// TIA Portal project "Styringsenhed" (V13)

(* hardware
DEVICE "S7-1200 station_1"  S7-1200 Station
   slot 0: "Rack_0"  Rack  V1.0
   slot 1: "PLC_1"  CPU 1214C DC/DC/DC  6ES7 214-1AG40-0XB0  V4.1
   slot 3: "AQ 1x12BIT_1"  6ES7 232-4HA30-0XB0  V1.0
DEVICE "HMI_1"  KTP600 Basic color PN
   slot 0: "HMI"  HMI  6AV6 647-0AD11-3AX0  12.0.0.0
   slot 1: "HMI_RT_1"  KTP600 Basic color PN  6AV6 647-0AD11-3AX0  12.0.0.0
   slot 5: "HMI_1.IE_CP_1"  PROFINET Interface
      slot 1: "PROFINET Interface_1"  PROFINET Interface
         slot 1: "Port_1"  Port
*)

// ===== PLC "PLC_1"  CPU 1214C DC/DC/DC =====

VAR_GLOBAL   // PLC tag table "Default tag table"
   "Trin1" AT %Q0.6 : Bool;
   "Trin2" AT %Q0.7 : Bool;
   "Trin3" AT %Q1.0 : Bool;
   "Trin4" AT %Q1.1 : Bool;
   "SpændingCentral" AT %MB0 : USInt;
   "ManuelMode" AT %I0.0 : Bool;
   "KnapOp" AT %I0.1 : Bool;
   "KnapNed" AT %I0.2 : Bool;
END_VAR

DATA_BLOCK "Trinskifter_DB"   // DB8
{ S7_Optimized_Access := 'FALSE' }
VERSION : 0.1
// stored: InstanceOfName Trinskifter
"Trinskifter"
BEGIN
END_DATA_BLOCK

// folder: System blocks/Program resources

DATA_BLOCK "ManTrinskift1til2"   // DB1
{ S7_Optimized_Access := 'FALSE' }
AUTHOR : Simatic
FAMILY : IEC
NAME : IEC_TMR
VERSION : 1.0
// stored: InstanceOfName ?
"?"
BEGIN
END_DATA_BLOCK

DATA_BLOCK "Trinskift2til1"   // DB2
{ S7_Optimized_Access := 'FALSE' }
AUTHOR : Simatic
FAMILY : IEC
NAME : IEC_TMR
VERSION : 1.0
// stored: InstanceOfName ?
"?"
BEGIN
END_DATA_BLOCK

DATA_BLOCK "Trinskift2til3"   // DB3
{ S7_Optimized_Access := 'FALSE' }
AUTHOR : Simatic
FAMILY : IEC
NAME : IEC_TMR
VERSION : 1.0
// stored: InstanceOfName ?
"?"
BEGIN
END_DATA_BLOCK

DATA_BLOCK "Trinskift1til2"   // DB4
{ S7_Optimized_Access := 'FALSE' }
AUTHOR : Simatic
FAMILY : IEC
NAME : IEC_TMR
VERSION : 1.0
// stored: InstanceOfName ?
"?"
BEGIN
END_DATA_BLOCK

DATA_BLOCK "Trinskift3til2"   // DB5
{ S7_Optimized_Access := 'FALSE' }
AUTHOR : Simatic
FAMILY : IEC
NAME : IEC_TMR
VERSION : 1.0
// stored: InstanceOfName ?
"?"
BEGIN
END_DATA_BLOCK

DATA_BLOCK "Trinskift3til4"   // DB6
{ S7_Optimized_Access := 'FALSE' }
AUTHOR : Simatic
FAMILY : IEC
NAME : IEC_TMR
VERSION : 1.0
// stored: InstanceOfName ?
"?"
BEGIN
END_DATA_BLOCK

DATA_BLOCK "Trinskift4til3"   // DB7
{ S7_Optimized_Access := 'FALSE' }
AUTHOR : Simatic
FAMILY : IEC
NAME : IEC_TMR
VERSION : 1.0
// stored: InstanceOfName ?
"?"
BEGIN
END_DATA_BLOCK

DATA_BLOCK "ManTrinskift2til3"   // DB9
{ S7_Optimized_Access := 'FALSE' }
AUTHOR : Simatic
FAMILY : IEC
NAME : IEC_TMR
VERSION : 1.0
// stored: InstanceOfName ?
"?"
BEGIN
END_DATA_BLOCK

DATA_BLOCK "ManTrinskift2til1"   // DB10
{ S7_Optimized_Access := 'FALSE' }
AUTHOR : Simatic
FAMILY : IEC
NAME : IEC_TMR
VERSION : 1.0
// stored: InstanceOfName ?
"?"
BEGIN
END_DATA_BLOCK

DATA_BLOCK "ManTrinskift3til4"   // DB11
{ S7_Optimized_Access := 'FALSE' }
AUTHOR : Simatic
FAMILY : IEC
NAME : IEC_TMR
VERSION : 1.0
// stored: InstanceOfName ?
"?"
BEGIN
END_DATA_BLOCK

DATA_BLOCK "ManTrinskift3til2"   // DB12
{ S7_Optimized_Access := 'FALSE' }
AUTHOR : Simatic
FAMILY : IEC
NAME : IEC_TMR
VERSION : 1.0
// stored: InstanceOfName ?
"?"
BEGIN
END_DATA_BLOCK

DATA_BLOCK "ManTrinskift4til3"   // DB13
{ S7_Optimized_Access := 'FALSE' }
AUTHOR : Simatic
FAMILY : IEC
NAME : IEC_TMR
VERSION : 1.0
// stored: InstanceOfName ?
"?"
BEGIN
END_DATA_BLOCK

// folder: (top level)

FUNCTION_BLOCK "Trinskifter"   // FB1, LAD
{ S7_Optimized_Access := 'FALSE' }
VERSION : 0.1
   VAR_TEMP   // added for the SCL form of the ladder/FBD networks
      _w1 : Bool;
      _w2 : Bool;
   END_VAR
BEGIN

REGION Network 1: Start
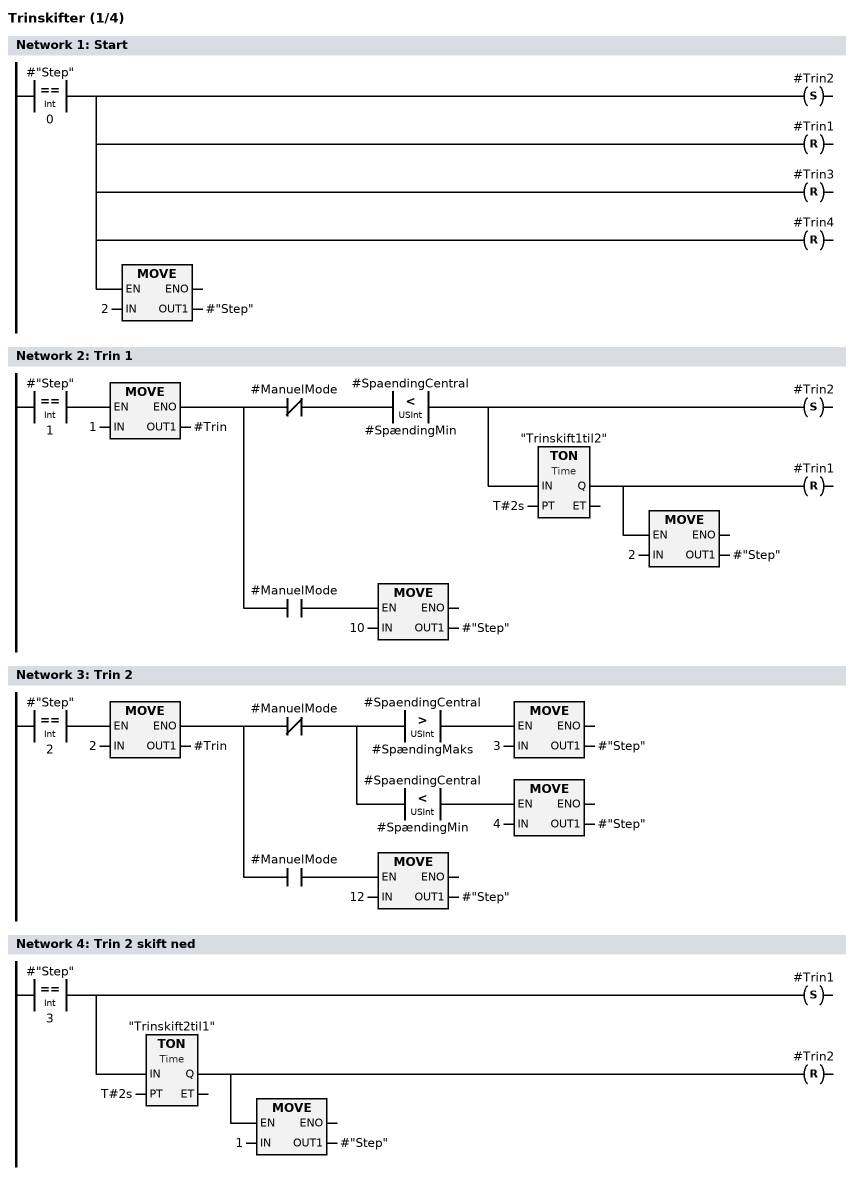
   RUNG wire#powerrail
      { S7_Templates := "SrcType := Int" } EQ_Contact(in1 := #"Step", in2 := 0)
      wire#w1
      S_Coil( #Trin2 )
   END_RUNG
   RUNG wire#w1
      R_Coil( #Trin1 )
   END_RUNG
   RUNG wire#w1
      R_Coil( #Trin3 )
   END_RUNG
   RUNG wire#w1
      R_Coil( #Trin4 )
   END_RUNG
   RUNG wire#w1
      Move(in := 2, out1 => #"Step")
   END_RUNG
   // the same network as SCL:
   IF #"Step" = 0 THEN
       #Trin2 := TRUE;
       #Trin1 := FALSE;
       #Trin3 := FALSE;
       #Trin4 := FALSE;
       #"Step" := 2;
   END_IF;
END_REGION

REGION Network 2: Trin 1
   #_w1 := #"Step" = 1;
   IF #_w1 THEN #Trin := 1; END_IF;
   #_w2 := #_w1 AND NOT #ManuelMode AND (#SpaendingCentral < #SpændingMin);
   IF #_w2 THEN #Trin2 := TRUE; END_IF;
   "Trinskift1til2".TON(IN := #_w2, PT := T#2s);
   IF "Trinskift1til2".Q THEN
       #Trin1 := FALSE;
       #"Step" := 2;
   END_IF;
   IF #_w1 AND #ManuelMode THEN #"Step" := 10; END_IF;
END_REGION

REGION Network 3: Trin 2
   RUNG wire#powerrail
      { S7_Templates := "SrcType := Int" } EQ_Contact(in1 := #"Step", in2 := 2)
      Move(in := 2, out1 => #Trin)
      wire#w1
      I_Contact( #ManuelMode )
      wire#w2
      { S7_Templates := "SrcType := USInt" } GT_Contact(in1 := #SpaendingCentral, in2 := #SpændingMaks)
      Move(in := 3, out1 => #"Step")
   END_RUNG
   RUNG wire#w2
      { S7_Templates := "SrcType := USInt" } LT_Contact(in1 := #SpaendingCentral, in2 := #SpændingMin)
      Move(in := 4, out1 => #"Step")
   END_RUNG
   RUNG wire#w1
      Contact( #ManuelMode )
      Move(in := 12, out1 => #"Step")
   END_RUNG
   // the same network as SCL:
   #_w1 := #"Step" = 2;
   IF #_w1 THEN #Trin := 2; END_IF;
   #_w2 := #_w1 AND NOT #ManuelMode;
   IF #_w2 AND (#SpaendingCentral > #SpændingMaks) THEN #"Step" := 3; END_IF;
   IF #_w2 AND (#SpaendingCentral < #SpændingMin) THEN #"Step" := 4; END_IF;
   IF #_w1 AND #ManuelMode THEN #"Step" := 12; END_IF;
END_REGION

REGION Network 4: Trin 2 skift ned
   #_w1 := #"Step" = 3;
   IF #_w1 THEN #Trin1 := TRUE; END_IF;
   "Trinskift2til1".TON(IN := #_w1, PT := T#2s);
   IF "Trinskift2til1".Q THEN
       #Trin2 := FALSE;
       #"Step" := 1;
   END_IF;
END_REGION

REGION Network 5: Trin 2 skift op
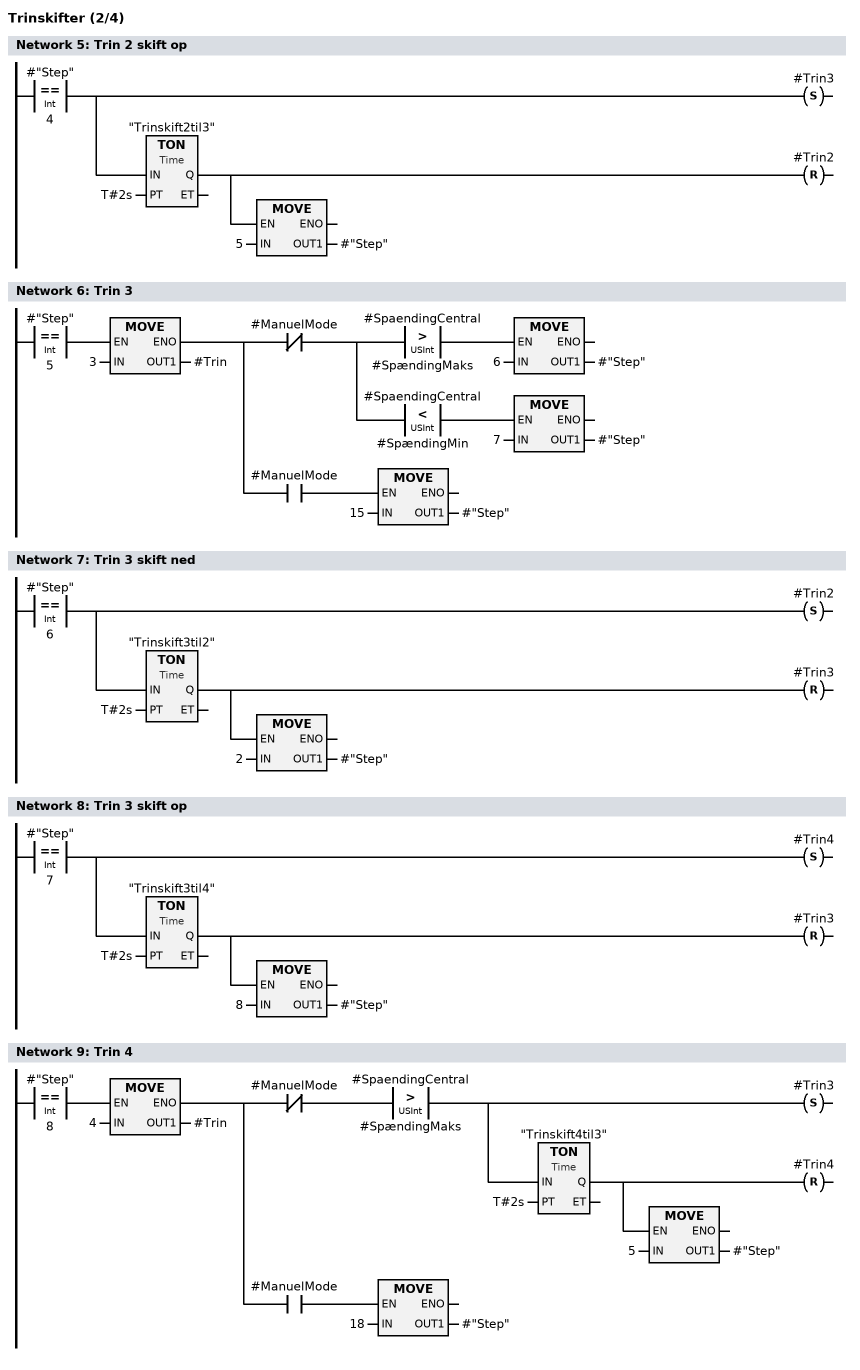
   #_w1 := #"Step" = 4;
   IF #_w1 THEN #Trin3 := TRUE; END_IF;
   "Trinskift2til3".TON(IN := #_w1, PT := T#2s);
   IF "Trinskift2til3".Q THEN
       #Trin2 := FALSE;
       #"Step" := 5;
   END_IF;
END_REGION

REGION Network 6: Trin 3
   RUNG wire#powerrail
      { S7_Templates := "SrcType := Int" } EQ_Contact(in1 := #"Step", in2 := 5)
      Move(in := 3, out1 => #Trin)
      wire#w1
      I_Contact( #ManuelMode )
      wire#w2
      { S7_Templates := "SrcType := USInt" } GT_Contact(in1 := #SpaendingCentral, in2 := #SpændingMaks)
      Move(in := 6, out1 => #"Step")
   END_RUNG
   RUNG wire#w2
      { S7_Templates := "SrcType := USInt" } LT_Contact(in1 := #SpaendingCentral, in2 := #SpændingMin)
      Move(in := 7, out1 => #"Step")
   END_RUNG
   RUNG wire#w1
      Contact( #ManuelMode )
      Move(in := 15, out1 => #"Step")
   END_RUNG
   // the same network as SCL:
   #_w1 := #"Step" = 5;
   IF #_w1 THEN #Trin := 3; END_IF;
   #_w2 := #_w1 AND NOT #ManuelMode;
   IF #_w2 AND (#SpaendingCentral > #SpændingMaks) THEN #"Step" := 6; END_IF;
   IF #_w2 AND (#SpaendingCentral < #SpændingMin) THEN #"Step" := 7; END_IF;
   IF #_w1 AND #ManuelMode THEN #"Step" := 15; END_IF;
END_REGION

REGION Network 7: Trin 3 skift ned
   #_w1 := #"Step" = 6;
   IF #_w1 THEN #Trin2 := TRUE; END_IF;
   "Trinskift3til2".TON(IN := #_w1, PT := T#2s);
   IF "Trinskift3til2".Q THEN
       #Trin3 := FALSE;
       #"Step" := 2;
   END_IF;
END_REGION

REGION Network 8: Trin 3 skift op
   #_w1 := #"Step" = 7;
   IF #_w1 THEN #Trin4 := TRUE; END_IF;
   "Trinskift3til4".TON(IN := #_w1, PT := T#2s);
   IF "Trinskift3til4".Q THEN
       #Trin3 := FALSE;
       #"Step" := 8;
   END_IF;
END_REGION

REGION Network 9: Trin 4
   #_w1 := #"Step" = 8;
   IF #_w1 THEN #Trin := 4; END_IF;
   #_w2 := #_w1 AND NOT #ManuelMode AND (#SpaendingCentral > #SpændingMaks);
   IF #_w2 THEN #Trin3 := TRUE; END_IF;
   "Trinskift4til3".TON(IN := #_w2, PT := T#2s);
   IF "Trinskift4til3".Q THEN
       #Trin4 := FALSE;
       #"Step" := 5;
   END_IF;
   IF #_w1 AND #ManuelMode THEN #"Step" := 18; END_IF;
END_REGION

REGION Network 10: Manuel trin 1
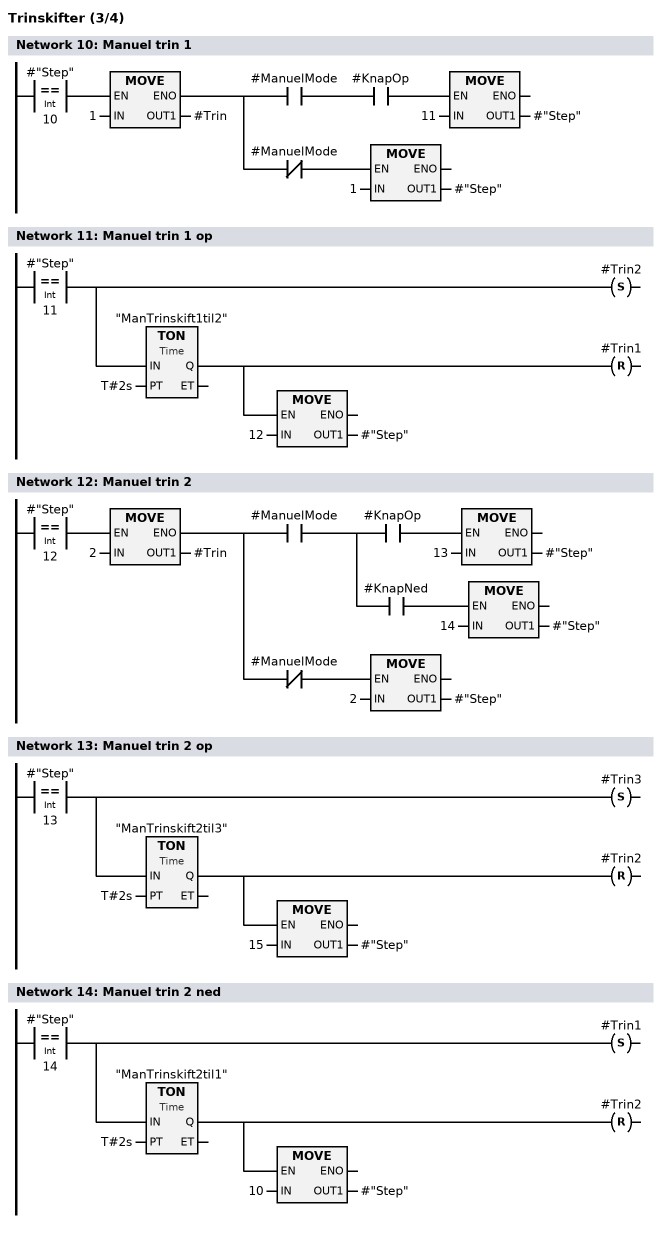
   RUNG wire#powerrail
      { S7_Templates := "SrcType := Int" } EQ_Contact(in1 := #"Step", in2 := 10)
      Move(in := 1, out1 => #Trin)
      wire#w1
      Contact( #ManuelMode )
      Contact( #KnapOp )
      Move(in := 11, out1 => #"Step")
   END_RUNG
   RUNG wire#w1
      I_Contact( #ManuelMode )
      Move(in := 1, out1 => #"Step")
   END_RUNG
   // the same network as SCL:
   #_w1 := #"Step" = 10;
   IF #_w1 THEN #Trin := 1; END_IF;
   IF #_w1 AND #ManuelMode AND #KnapOp THEN #"Step" := 11; END_IF;
   IF #_w1 AND NOT #ManuelMode THEN #"Step" := 1; END_IF;
END_REGION

REGION Network 11: Manuel trin 1 op
   #_w1 := #"Step" = 11;
   IF #_w1 THEN #Trin2 := TRUE; END_IF;
   "ManTrinskift1til2".TON(IN := #_w1, PT := T#2s);
   IF "ManTrinskift1til2".Q THEN
       #Trin1 := FALSE;
       #"Step" := 12;
   END_IF;
END_REGION

REGION Network 12: Manuel trin 2
   RUNG wire#powerrail
      { S7_Templates := "SrcType := Int" } EQ_Contact(in1 := #"Step", in2 := 12)
      Move(in := 2, out1 => #Trin)
      wire#w1
      Contact( #ManuelMode )
      wire#w2
      Contact( #KnapOp )
      Move(in := 13, out1 => #"Step")
   END_RUNG
   RUNG wire#w2
      Contact( #KnapNed )
      Move(in := 14, out1 => #"Step")
   END_RUNG
   RUNG wire#w1
      I_Contact( #ManuelMode )
      Move(in := 2, out1 => #"Step")
   END_RUNG
   // the same network as SCL:
   #_w1 := #"Step" = 12;
   IF #_w1 THEN #Trin := 2; END_IF;
   #_w2 := #_w1 AND #ManuelMode;
   IF #_w2 AND #KnapOp THEN #"Step" := 13; END_IF;
   IF #_w2 AND #KnapNed THEN #"Step" := 14; END_IF;
   IF #_w1 AND NOT #ManuelMode THEN #"Step" := 2; END_IF;
END_REGION

REGION Network 13: Manuel trin 2 op
   #_w1 := #"Step" = 13;
   IF #_w1 THEN #Trin3 := TRUE; END_IF;
   "ManTrinskift2til3".TON(IN := #_w1, PT := T#2s);
   IF "ManTrinskift2til3".Q THEN
       #Trin2 := FALSE;
       #"Step" := 15;
   END_IF;
END_REGION

REGION Network 14: Manuel trin 2 ned
   #_w1 := #"Step" = 14;
   IF #_w1 THEN #Trin1 := TRUE; END_IF;
   "ManTrinskift2til1".TON(IN := #_w1, PT := T#2s);
   IF "ManTrinskift2til1".Q THEN
       #Trin2 := FALSE;
       #"Step" := 10;
   END_IF;
END_REGION

REGION Network 15: Manuel trin 3
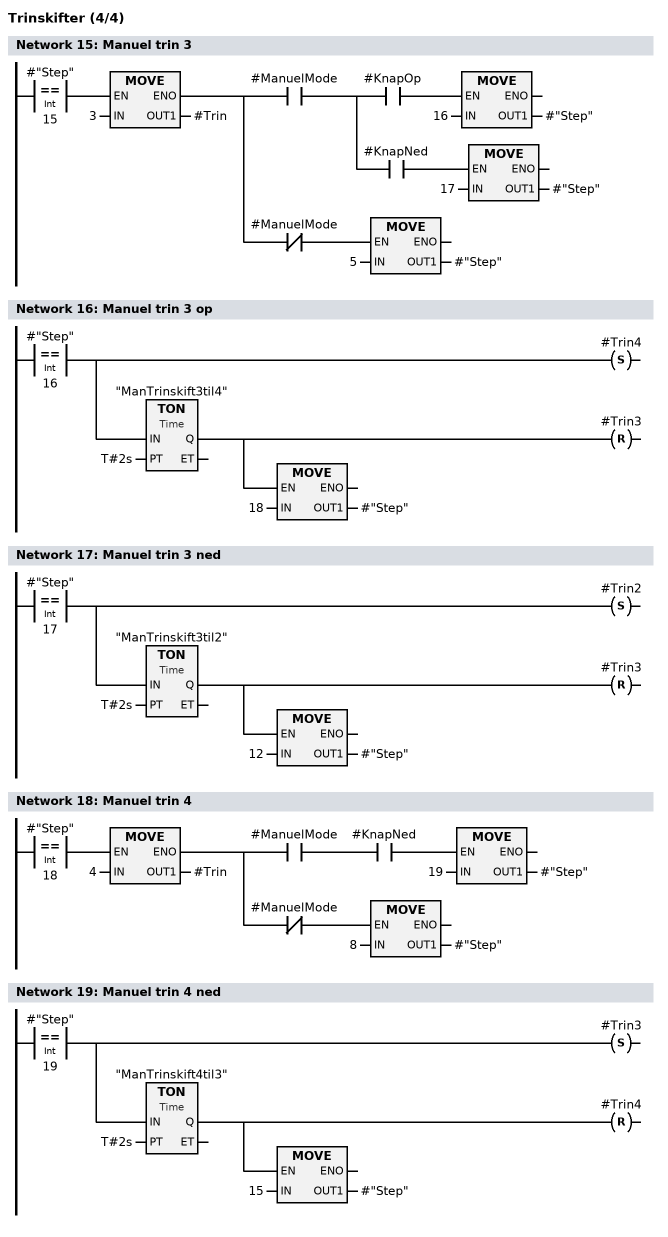
   RUNG wire#powerrail
      { S7_Templates := "SrcType := Int" } EQ_Contact(in1 := #"Step", in2 := 15)
      Move(in := 3, out1 => #Trin)
      wire#w1
      Contact( #ManuelMode )
      wire#w2
      Contact( #KnapOp )
      Move(in := 16, out1 => #"Step")
   END_RUNG
   RUNG wire#w2
      Contact( #KnapNed )
      Move(in := 17, out1 => #"Step")
   END_RUNG
   RUNG wire#w1
      I_Contact( #ManuelMode )
      Move(in := 5, out1 => #"Step")
   END_RUNG
   // the same network as SCL:
   #_w1 := #"Step" = 15;
   IF #_w1 THEN #Trin := 3; END_IF;
   #_w2 := #_w1 AND #ManuelMode;
   IF #_w2 AND #KnapOp THEN #"Step" := 16; END_IF;
   IF #_w2 AND #KnapNed THEN #"Step" := 17; END_IF;
   IF #_w1 AND NOT #ManuelMode THEN #"Step" := 5; END_IF;
END_REGION

REGION Network 16: Manuel trin 3 op
   #_w1 := #"Step" = 16;
   IF #_w1 THEN #Trin4 := TRUE; END_IF;
   "ManTrinskift3til4".TON(IN := #_w1, PT := T#2s);
   IF "ManTrinskift3til4".Q THEN
       #Trin3 := FALSE;
       #"Step" := 18;
   END_IF;
END_REGION

REGION Network 17: Manuel trin 3 ned
   #_w1 := #"Step" = 17;
   IF #_w1 THEN #Trin2 := TRUE; END_IF;
   "ManTrinskift3til2".TON(IN := #_w1, PT := T#2s);
   IF "ManTrinskift3til2".Q THEN
       #Trin3 := FALSE;
       #"Step" := 12;
   END_IF;
END_REGION

REGION Network 18: Manuel trin 4
   RUNG wire#powerrail
      { S7_Templates := "SrcType := Int" } EQ_Contact(in1 := #"Step", in2 := 18)
      Move(in := 4, out1 => #Trin)
      wire#w1
      Contact( #ManuelMode )
      Contact( #KnapNed )
      Move(in := 19, out1 => #"Step")
   END_RUNG
   RUNG wire#w1
      I_Contact( #ManuelMode )
      Move(in := 8, out1 => #"Step")
   END_RUNG
   // the same network as SCL:
   #_w1 := #"Step" = 18;
   IF #_w1 THEN #Trin := 4; END_IF;
   IF #_w1 AND #ManuelMode AND #KnapNed THEN #"Step" := 19; END_IF;
   IF #_w1 AND NOT #ManuelMode THEN #"Step" := 8; END_IF;
END_REGION

REGION Network 19: Manuel trin 4 ned
   #_w1 := #"Step" = 19;
   IF #_w1 THEN #Trin3 := TRUE; END_IF;
   "ManTrinskift4til3".TON(IN := #_w1, PT := T#2s);
   IF "ManTrinskift4til3".Q THEN
       #Trin4 := FALSE;
       #"Step" := 15;
   END_IF;
END_REGION
END_FUNCTION_BLOCK

ORGANIZATION_BLOCK "Main"   // OB1, LAD, ProgramCycle
TITLE = "Main Program Sweep (Cycle)"
{ S7_Optimized_Access := 'FALSE' }
VERSION : 0.1
BEGIN

REGION Network 1
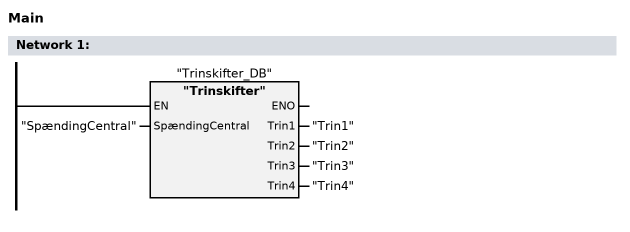
   RUNG wire#powerrail
      "Trinskifter_DB"(SpændingCentral := "SpændingCentral", Trin1 => "Trin1", Trin2 => "Trin2", Trin3 => "Trin3", Trin4 => "Trin4")
   END_RUNG
   // the same network as SCL:
   "Trinskifter_DB"(SpændingCentral := "SpændingCentral",   // "Trinskifter"
                    Trin1 => "Trin1",
                    Trin2 => "Trin2",
                    Trin3 => "Trin3",
                    Trin4 => "Trin4");
END_REGION
END_ORGANIZATION_BLOCK